// TIA Portal V20 export
DATA_BLOCK "BK08"   // DB203
// stored: MemoryReserve 100
   VAR
      "X10-1 UW ELECTRODE FIX LEFT TOP V/C ON" : Bool;
      "X10-2 UW ELECTRODE FIX LEFT TOP V/C OFF" : Bool;
      "X12-1 UW ELECTRODE FIX LEFT BTM V/C ON" : Bool;
      "X12-2 UW ELECTRODE FIX LEFT BTM V/C OFF" : Bool;
      "X14-1 UW ELECTRODE FIX RIGHT TOP V/C ON" : Bool;
      "X14-2 UW ELECTRODE FIX RIGHT TOP V/C OFF" : Bool;
      "X16-1 UW ELECTRODE FIX RIGHT BTM V/C ON" : Bool;
      "X16-2 UW ELECTRODE FIX RIGHT BTM V/C OFF" : Bool;
   END_VAR
BEGIN
END_DATA_BLOCK
